// TIA Portal V19 export
FUNCTION "LAF_GetCycleTimes" : Void   // FC81, LAD
TITLE = LAF_GetCycleTimes
AUTHOR : Siemens Digital Industries
FAMILY : LAF
VERSION : 1.2
// This blocks monitors the current, maximum and minimum cycle times of the PLC.
// stored: Access Published, IsIECCheckEnabled true, SetENOAutomatically false
   VAR_IN_OUT
      reset : Bool;   // Reset max / min cycle time
      prevCycle : UInt;   // Previous cycle time
      maxCycle : UInt;   // Maximum cycle time
      minCycle : UInt;   // Minimum cycle time
   END_VAR
   VAR_TEMP
      tempStndPrevCycle : LTime;   // Current plc cycle time / Aktuelle CPU Zykluszeit
      tempRetVal1 : Int;   // Ret_Val / Rückgabewert
      tempUlint : ULInt;   // Temp UInt / Temporär UInt
      tempReal : ULInt;   // Temp Real / Temporär Real
   END_VAR
   VAR_TEMP   // added for the SCL form of the ladder/FBD networks
      _w1 : Bool;
   END_VAR
BEGIN

REGION Network 1: BLOCK INFO HEADER
   // SIEMENS AG / (c)Copyright 2024
   // ------------------------------------------------------------------------------
   // Title:            LAF_GetCycleLimits
   // Comment/Function: This blocks monitors the current, maximum and minimum cycle times of the PLC.
   // Library/Family:   Library of Automation Framework
   // Author:                Siemens Digital Industry
   // Tested with:       S7-PLCSIM Advanced 6.0
   // Engineering:      TIA Portal V19
   // Restrictions:       ---
   // Requirements:   ---
   // ------------------------------------------------------------------------------
   // Change log table:
   // Version  | Date       | Expert in charge       | Changes applied
   // ---------|------------|------------------------|------------------------------
   // 01.01.00 | 21.06.2024 | SIMATIC Systems Support
   //                         First released version
   // 01.02.00 | 30.09.2024 | SIMATIC Systems Support
   //                         Block information properties updated
END_REGION

REGION Network 2: DESCRIPTION
   // This block monitors the cycle times of the PLC, recording the current, maximum and minimum values of the cycle times, and allows resetting these values through a reset signal.
END_REGION

REGION Network 3: Read cycle time of previous cycle / Zyklus Zeiten
   // Berechnung der minimalen, maximalen und vorherigen bzw. aktuellen Zykluszeit
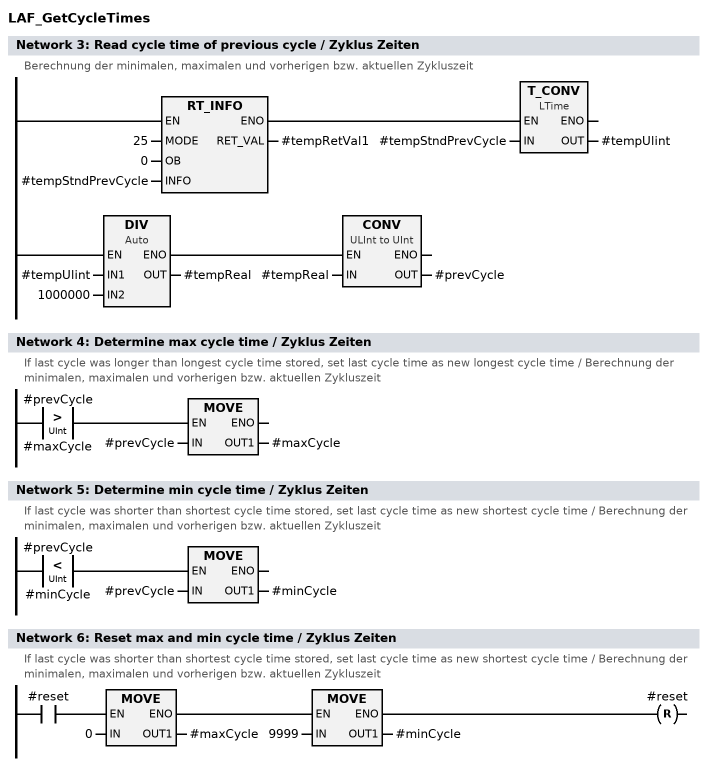
   RUNG wire#powerrail
      RT_INFO(MODE := 25, OB := 0, INFO := #tempStndPrevCycle, Ret_Val => #tempRetVal1)
      { S7_Templates := "[src_type := LTime, dest_type := ULInt]" } T_CONV(IN := #tempStndPrevCycle, OUT => #tempUlint)
   END_RUNG
   RUNG wire#powerrail
      Div(in1 := #tempUlint, in2 := 1000000, out => #tempReal)
      { S7_Templates := "[SrcType := ULInt, DestType := UInt]" } Convert(in := #tempReal, out => #prevCycle)
   END_RUNG
   // the same network as SCL:
   #tempRetVal1 := RT_INFO(MODE := 25, OB := 0, INFO := #tempStndPrevCycle, ENO => #_w1);
   IF #_w1 THEN T_CONV(IN := #tempStndPrevCycle, OUT => #tempUlint); END_IF;
   #tempReal := #tempUlint / 1000000;
   #prevCycle := ULINT_TO_UINT(#tempReal);
END_REGION

REGION Network 4: Determine max cycle time / Zyklus Zeiten
   // If last cycle was longer than longest cycle time stored, set last cycle time as new longest cycle time / Berechnung der minimalen, maximalen und vorherigen bzw. aktuellen Zykluszeit
   RUNG wire#powerrail
      { S7_Templates := "SrcType := UInt" } GT_Contact(in1 := #prevCycle, in2 := #maxCycle)
      Move(in := #prevCycle, out1 => #maxCycle)
   END_RUNG
   // the same network as SCL:
   IF #prevCycle > #maxCycle THEN #maxCycle := #prevCycle; END_IF;
END_REGION

REGION Network 5: Determine min cycle time / Zyklus Zeiten
   // If last cycle was shorter than shortest cycle time stored, set last cycle time as new shortest cycle time / Berechnung der minimalen, maximalen und vorherigen bzw. aktuellen Zykluszeit
   RUNG wire#powerrail
      { S7_Templates := "SrcType := UInt" } LT_Contact(in1 := #prevCycle, in2 := #minCycle)
      Move(in := #prevCycle, out1 => #minCycle)
   END_RUNG
   // the same network as SCL:
   IF #prevCycle < #minCycle THEN #minCycle := #prevCycle; END_IF;
END_REGION

REGION Network 6: Reset max and min cycle time / Zyklus Zeiten
   // If last cycle was shorter than shortest cycle time stored, set last cycle time as new shortest cycle time / Berechnung der minimalen, maximalen und vorherigen bzw. aktuellen Zykluszeit
   RUNG wire#powerrail
      Contact( #reset )
      Move(in := 0, out1 => #maxCycle)
      Move(in := 9999, out1 => #minCycle)
      R_Coil( #reset )
   END_RUNG
   // the same network as SCL:
   IF #reset THEN
       #maxCycle := 0;
       #minCycle := 9999;
       #reset := FALSE;
   END_IF;
END_REGION
END_FUNCTION
